// SIMATIC S7-200 SMART project (STEP 7-Micro/WIN SMART), CPU ST40

SYMBOL_TABLE 表格 1
报警红灯             Q0.1     // 严重故障报警指示
复位按钮             I0.4     // 手动复位按钮
故障计数器            C0       // 严重故障累计次数
故障确认定时器          T37      // 严重故障延时3秒确认
滚动体故障            I0.3     // CNN诊断-滚动体故障信号
内圈故障             I0.1     // CNN诊断-内圈故障信号
频繁报警             Q0.3     // 故障超过5次输出
停机保护             Q0.2     // 电机停机保护继电器
外圈故障             I0.2     // CNN诊断-外圈故障信号
预警黄灯             Q0.0     // 轻度故障预警指示
END_SYMBOL_TABLE

ORGANIZATION_BLOCK MAIN:OB1
TITLE=程序注释
BEGIN
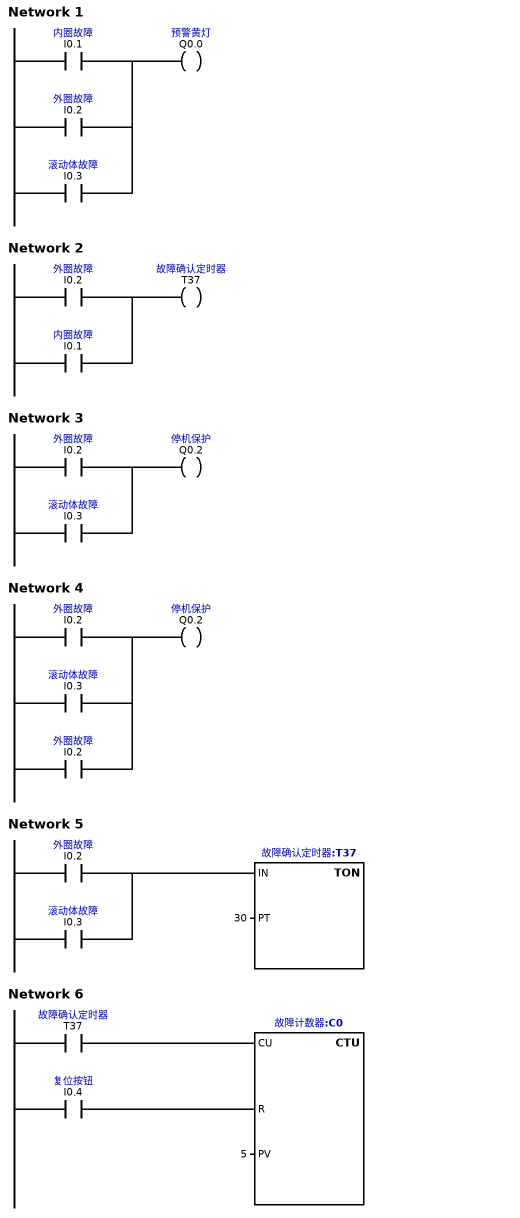
Network 1
LD     内圈故障:I0.1
O      外圈故障:I0.2
O      滚动体故障:I0.3
=      预警黄灯:Q0.0
Network 2
LD     外圈故障:I0.2
O      内圈故障:I0.1
=      故障确认定时器:T37
Network 3
LD     外圈故障:I0.2
O      滚动体故障:I0.3
=      停机保护:Q0.2
Network 4
LD     外圈故障:I0.2
O      滚动体故障:I0.3
O      外圈故障:I0.2
=      停机保护:Q0.2
Network 5
LD     外圈故障:I0.2
O      滚动体故障:I0.3
TON    故障确认定时器:T37, 30
Network 6
LD     故障确认定时器:T37
LD     复位按钮:I0.4
CTU    故障计数器:C0, 5
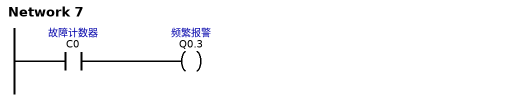
Network 7
LD     故障计数器:C0
=      频繁报警:Q0.3
END_ORGANIZATION_BLOCK

// SBR2: protected block, not included
